FUNCTION_BLOCK CL_CardCom EXTENDS CL_MasterRootClass
VAR
  //private internal methods
  bComInit       : BOOL := FALSE;
  _stCardState_P : POINTER TO ST_CardState_HWI;
END_VAR

IF bComInit THEN
  THIS^.RunCom();
END_IF

METHOD InitCom : BOOL
VAR_INPUT
  stCardStateIn_P : POINTER TO ST_CardState_HWI;
END_VAR
InitCom := false;
_stCardState_P  := stCardStateIn_P;
IF _stCardState_P <> 0 AND NOT bComInit THEN
  bComInit := InitCom := InitDefectCom();
END_IF
END_METHOD

METHOD PROTECTED InitDefectCom : BOOL
VAR_INPUT
END_VAR
InitDefectCom := true;
END_METHOD

METHOD PRIVATE RunCom
VAR_INPUT
END_VAR
END_METHOD

END_FUNCTION_BLOCK

(* stored: Version 1.1.0.1, ProductVersion 3.1.4024.12
   POU CL_CardCom: Id {b34a7690-b9a4-4b52-9d49-bc4d03a2a3f1}, SpecialFunc None
   Method InitCom: Id {676f847c-dc14-4be2-9aee-701fde478720}
   Method InitDefectCom: Id {136eb99c-79aa-4a5e-8ff5-24101f70345f}
   Method RunCom: Id {283a85d4-cf26-4be0-afc9-b81468d2ed47} *)
